(* Schneider Machine Expert - Basic project Ex1TM221, file version 1.8.0.0 *)
(* ProjectInformations: Name=New project *)

HARDWARE
  Cpu 0: TM221CE16R
  EthernetConfiguration: NetworkName=M221, IpAllocationMode=FixedAddress, IpAddress=192.168.1.22, SubnetMask=255.255.255.0
  SerialLineConfiguration: Baud=Baud19200, Parity=ParityEven, DataBits=DataBits8, StopBits=StopBits1, PhysicalMedium=PhysicalMediumRs485, TransmissionMode=TransmissionModeModbusRtu, SlaveId=1, Addressing=SlaveAddressing
  MastTask: UsePeriodScanMode=false, PeriodScan=100
  FastTask: Period=255
  CpuBehavior: StartingMode=StartAsPreviousState, AutoSaveRamOnEeprom=true, WatchdogPeriod=250

SYMBOLS  (address, symbol, comment, settings)

POU input
  (* SectionNumber=1 *)

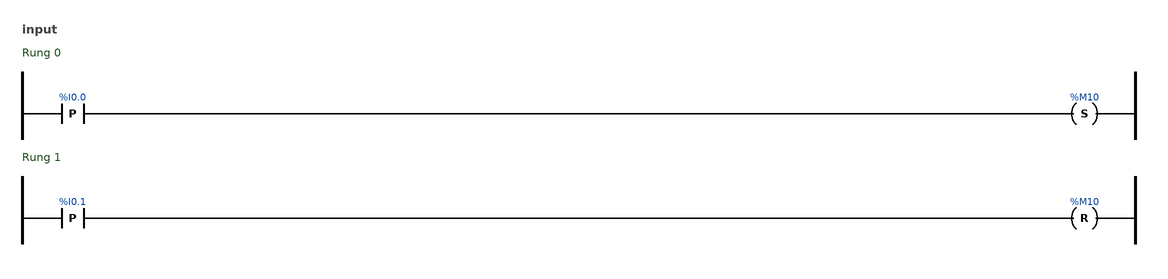

// Rung 0
  LDR %I0.0
  S %M10
  // as ST:
  //   IF RISING(%I0.0) THEN %M10 := TRUE; END_IF;

// Rung 1
  LDR %I0.1
  R %M10
  // as ST:
  //   IF RISING(%I0.1) THEN %M10 := FALSE; END_IF;

POU output
  (* SectionNumber=2 *)

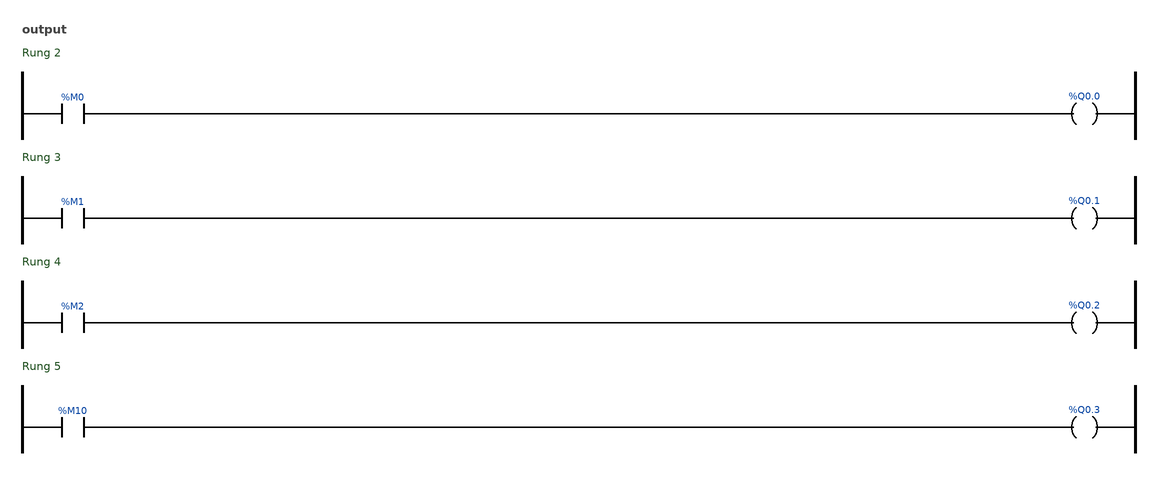

// Rung 2
  LD %M0
  ST %Q0.0
  // as ST:
  //   %Q0.0 := %M0;

// Rung 3
  LD %M1
  ST %Q0.1
  // as ST:
  //   %Q0.1 := %M1;

// Rung 4
  LD %M2
  ST %Q0.2
  // as ST:
  //   %Q0.2 := %M2;

// Rung 5
  LD %M10
  ST %Q0.3
  // as ST:
  //   %Q0.3 := %M10;
